FUNCTION_BLOCK AD_SHL (* FB to calculate bitwise SHL (generic FB) *)
  (* Standard: 61499-2; Description: Copyright (c) 2026 HR Agrartechnik GmbH This program and the accompanying materials are made available under the terms of the Eclipse Public License 2.0 which is available at https://www.eclipse.org/legal/epl-2.0/ SPDX-License-Identifier: EPL-2.0 *)
  (* Version 1.1, 2026-04-20, Franz Höpfinger, HR Agrartechnik GmbH, Added UPDATE event for N to satisfy Basic FB / logic rules *)
  (* Version 1.0, 2026-04-20, Franz Höpfinger, HR Agrartechnik GmbH, initial API and implementation *)
  PACKAGE adapter::iec61131::bitwise;
  IMPORT eclipse4diac::core::TypeHash;
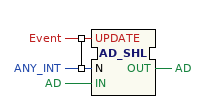
  EVENT_INPUT
    UPDATE WITH N; (* Update shift count *)
  END_EVENT
  VAR_INPUT
    N : ANY_INT; (* Number of bits to shift *)
  END_VAR
  SOCKETS
    IN : adapter::types::unidirectional::AD; (* SHL input *)
  END_SOCKETS
  PLUGS
    OUT : adapter::types::unidirectional::AD; (* SHL result *)
  END_PLUGS
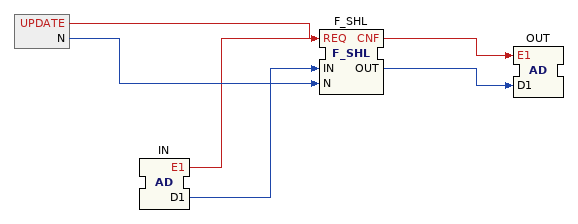
  FBS
    F_SHL : iec61131::bitwiseOperators::F_SHL;
  END_FBS
  EVENT_CONNECTIONS
    F_SHL.CNF TO OUT.E1;
    IN.E1 TO F_SHL.REQ;
    UPDATE TO F_SHL.REQ;
  END_CONNECTIONS
  DATA_CONNECTIONS
    F_SHL.OUT TO OUT.D1;
    IN.D1 TO F_SHL.IN;
    N TO F_SHL.N;
  END_CONNECTIONS
END_FUNCTION_BLOCK
